Staubli VAL3: socketServer.pjx

--- socketServer.pjx ---
Parameters version=s7.9.1 stackSize=5000 millimeterUnit=true
Program file=actGesture.pgx
Program file=actMovement.pgx
Program file=dataGet.pgx
Program file=detectInput.pgx
Program file=gestureFist.pgx
Program file=gestureSpread.pgx
Program file=gestureWaveIn.pgx
Program file=gestureWaveout.pgx
Program file=parseMovement.pgx
Program file=start.pgx
Program file=stop.pgx
Data file=socketServer.dtx

--- socketServer.dtx ---
bool bClawClosed = true
bool bDetectInput
bool bParseResult = true
jointRx home = {j1=0.299277, j2=90.551723, j3=0.116241, j4=-0.513613, j5=0.611835, j6=-177.732323}
jointRx homePoint = {j2=35, j6=-179}
jointRx jTest
jointRx joint1Test = {j2=3.0286646, j3=-0.380119, j4=-86.65991, j5=4.31054, j6=-179.150356}
jointRx joint1TestCopy = {j2=3.0286646, j3=-0.380119, j4=-86.65991, j5=4.31054, j6=-179.150356}
jointRx startPoint = {j2=29.71527, j3=59.600259, j4=-86.849417, j5=2.295044, j6=-178.473868}
jointRx waveIn = {j1=1.950737, j2=29.71527, j3=-3.0442775, j4=-86.849417, j5=2.295044, j6=-178.473868}
jointRx wristDown = {j1=1.747969, j2=68.569512, j3=20.407078, j4=-4.314453, j5=62.758443, j6=-270}
jointRx wristUp = {j1=1.747969, j2=68.569512, j3=20.407078, j4=-7.419285, j5=-49.114677, j6=-260.995824}
mdesc nom_speed = {rmax=9999, blend=off}
num nBuffer
num nFailCounter
num nIParseMovement
num nMovementData[3]
num nNum = -1
num nRXMovement = 70
num nTrsfJointArray[6]
  [0] = 11
  [1] = 3.0286646
  [2] = -0.380119
  [3] = -86.65991
  [4] = 4.31054
  [5] = -179.150356
num nXMovement = 11
num nZMovement = 168
pointRs pPointRs = {fatherId=world[0]}
pointRs pPointRs1 = {fatherId=world[0]}
sio sioSocket = {link=Socket\HelloServer}
string sBuffer
string sGetMovement
string sInput[50]
string sString = ")"
tool tClaw = {z=90, fatherId=flange[0], ioLink=valve1}
trsf trWorkingPoint
jointRx jJointRx = {j1=0.299277, j2=90.551723, j3=0.116241, j4=-0.513613, j5=0.611835, j6=-177.732323}
jointRx jJointRx1 = {j2=88.351928, j6=-179.151046}
jointRx homePointCopy = {j2=35, j6=-179}
num homePointArray[6]
  [1] = 35
  [5] = -179

--- start.pgx ---
public program start()
begin

  // The start function's purpose is to make sure everything is reset and setup
  // It starts by initing a few variables the program uses then moving the arm to the homePoint


  //initing a few variables
  nBuffer=0
  nNum=0
  nFailCounter=0
  bDetectInput=false
  sInput=""

  //Set the arm at the homePoint
  movej(homePoint,tClaw,nom_speed)
  waitEndMove()
  //call enablePowerTest()
  call detectInput()
end

--- actGesture.pgx ---
program actGesture()
begin
  //putln("GestureCalled")
  //putln(sInput)
  if (sInput=="fist")
    call gestureFist()
  elseIf (sInput=="waveIn")
    call gestureWaveIn()
  elseIf (sInput=="waveOut")
    call gestureWaveout()
  elseIf (sInput=="fingersSpread")
    call gestureSpread()
  endIf

end

--- actMovement.pgx ---
program actMovement()
begin
  putln(nXMovement)
  putln(nZMovement)
  putln(nRXMovement)

  if nXMovement > 80
    nXMovement = 80
  elseIf nXMovement < -80
    nXMovement = -80
  endIf

  if nZMovement > 80
    nZMovement = 80
  elseIf nZMovement < -80
    nZMovement = -80
  endIf

  if nRXMovement > 80
    nRXMovement = 80
  elseIf nRXMovement < -80
    nRXMovement = -80
  endIf

  homePointArray[0] = nXMovement
  homePointArray[2] = nZMovement
  homePointArray[3] = nRXMovement


  homePointCopy = {homePointArray[0],homePointArray[1],homePointArray[2],homePointArray[3],homePointArray[4],homePointArray[5]}

  movej(homePointCopy,tClaw,nom_speed)
  //waveIn[0] =
  //waveIn[1] =



end

--- dataGet.pgx ---
program dataGet()
begin
  //dataGet essentially gathers all of the inputs together and then calls the appropiate method
  //It is VITAL that the signal sent ends in either a ) (gesture) and } (movement).
  sBuffer=chr(nBuffer)
  //putln(sBuffer)
  if (sBuffer==")")
    //putln("dataGet")
    call actGesture()
    sInput=""
    nBuffer=0
    sBuffer=""
  elseIf (sBuffer=="}")
    //putln(sInput)
    call parseMovement()
    sInput=""
    nBuffer=0
    sBuffer=""
  else
    sInput=sInput+sBuffer
  endIf
  //sBuffer = ""
end

--- detectInput.pgx ---
program detectInput()
begin
  //Detect input detects if it is getting a signal and then calls the dataGet
  //method. Which creates the input. Since if I sent "hellWorld" through the client to the server. It would
  //be sent one character at a time. That is why we have the while loop. sioGet has a very useful function where it will
  //pause the entire program until it recieves a signal. Preventing the while loop from iterating.
  while true
    nNum=sioGet(sioSocket,nBuffer)
    //putln(nNum)
    if nNum>=0
      //putln("dataGet called")
      call dataGet()
    endIf
  endWhile
end

--- gestureFist.pgx ---
program gestureFist()
begin
  //close(tClaw)



  if (bClawClosed==false)
  close(tClaw)
  putln("Fist Closed")
  bClawClosed=true
  elseIf (bClawClosed==true)
  open(tClaw)
  putln("Fist Opened")
  bClawClosed=false
  endIf
end

--- gestureSpread.pgx ---
program gestureSpread()
begin
  //open(tClaw)
end

--- gestureWaveIn.pgx ---
program gestureWaveIn()
begin
  putln("WaveInCAlled")
  joint1TestCopy = joint1Test
  movej(joint1Test,tClaw,nom_speed)
end

--- gestureWaveout.pgx ---
program gestureWaveout()
begin
  putln("WaveOut Called")
  movej(wristUp,tClaw,nom_speed)
end

--- parseMovement.pgx ---
program parseMovement()
begin
  //putln(sInput)
  sGetMovement=sInput[0]

  sGetMovement=toNum(sGetMovement,nXMovement,bParseResult)
  sGetMovement=toNum(sGetMovement,nZMovement,bParseResult)
  sGetMovement=toNum(sGetMovement,nRXMovement,bParseResult)

  //putln(nXMovement)
  //putln(nZMovement)
  //putln(nRXMovement)

  call actMovement()
end

--- stop.pgx ---
program stop()
begin
  homePointCopy = homePoint
  popUpMsg("Pending movement commands have been canceled")
  resetMotion()
end
